(* PLC project mainPLC, Beckhoff Automation GmbH TwinCAT PLC Control 3.5.13.21 *)
(* stored: creationDateTime 2022-06-01T19:40:54.4880245, modificationDateTime 2022-06-01T19:40:54.4900208 *)

PROGRAM MAIN
VAR
	increment 	AT %I*	: INT 	:= 0;
	sum 		AT %Q*	: INT	:= 0;
END_VAR

            sum := sum + increment;
          
END_PROGRAM
